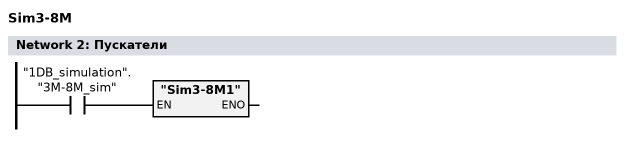
   RUNG wire#powerrail
      Contact( "1DB_simulation"."3M-8M_sim" )
      "Sim3-8M1"()
   END_RUNG
   // the same network as SCL:
   IF "1DB_simulation"."3M-8M_sim" THEN "Sim3-8M1"(); END_IF;
END_REGION
END_FUNCTION

FUNCTION "SimDym" : Void   // FC909, LAD
{ S7_Optimized_Access := 'TRUE' }
VERSION : 0.1
   VAR_TEMP
      trValue : Real;
      trValue_2 : Real;
      trValue_3 : Real;
   END_VAR
BEGIN

REGION Network 2: Скорость двигателя в %
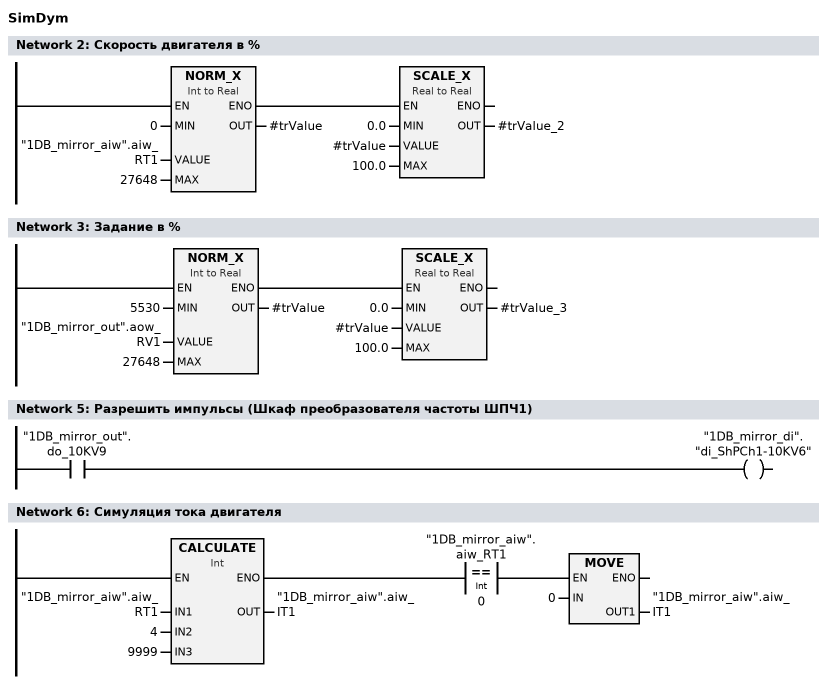
   RUNG wire#powerrail
      { S7_Templates := "[SrcType := Int, DestType := Real]" } Normalize(min := 0, value := "1DB_mirror_aiw".aiw_RT1, max := 27648, out => #trValue)
      { S7_Templates := "[SrcType := Real, DestType := Real]" } Scale(min := 0.0, value := #trValue, max := 100.0, out => #trValue_2)
   END_RUNG
   // the same network as SCL:
   #trValue := NORM_X(MIN := 0, VALUE := "1DB_mirror_aiw".aiw_RT1, MAX := 27648);
   #trValue_2 := SCALE_X(MIN := 0.0, VALUE := #trValue, MAX := 100.0);
END_REGION

REGION Network 3: Задание в %
   RUNG wire#powerrail
      { S7_Templates := "[SrcType := Int, DestType := Real]" } Normalize(min := 5530, value := "1DB_mirror_out".aow_RV1, max := 27648, out => #trValue)
      { S7_Templates := "[SrcType := Real, DestType := Real]" } Scale(min := 0.0, value := #trValue, max := 100.0, out => #trValue_3)
   END_RUNG
   // the same network as SCL:
   #trValue := NORM_X(MIN := 5530, VALUE := "1DB_mirror_out".aow_RV1, MAX := 27648);
   #trValue_3 := SCALE_X(MIN := 0.0, VALUE := #trValue, MAX := 100.0);
END_REGION

REGION Network 4 (SCL): Симуляция разгона и торможения
   //IF "1DB_mirror_out".do_1KV10 AND "1DB_mirror_out".do_1KV9
       //AND (NOT "HMI-Machinery".Dym.xSwitchAutoMode) THEN
   IF "1DB_mirror_out".aow_RV1 >0 THEN
       //IF #trValue_2 < "HMI-Machinery".Dym.rSpeedGoTo THEN
       IF #trValue_2 < #trValue_3 THEN
           "1DB_mirror_aiw".aiw_RT1 += 15;
       END_IF;
       IF #trValue_2 > #trValue_3 THEN
           "1DB_mirror_aiw".aiw_RT1 -= 19;
       END_IF;
   ELSE
       "1DB_mirror_aiw".aiw_RT1 := 0;
   END_IF;
END_REGION

REGION Network 5: Разрешить импульсы (Шкаф преобразователя частоты ШПЧ1)
   RUNG wire#powerrail
      Contact( "1DB_mirror_out".do_10KV9 )
      Coil( "1DB_mirror_di"."di_ShPCh1-10KV6" )
   END_RUNG
   // the same network as SCL:
   "1DB_mirror_di"."di_ShPCh1-10KV6" := "1DB_mirror_out".do_10KV9;
END_REGION

REGION Network 6: Симуляция тока двигателя
   RUNG wire#powerrail
      { S7_Templates := "SrcType := Int"; S7_Expression := "IN1/IN2 +IN3" } Calculate(in1 := "1DB_mirror_aiw".aiw_RT1, in2 := 4, in3 := 9999, out => "1DB_mirror_aiw".aiw_IT1)
      { S7_Templates := "SrcType := Int" } EQ_Contact(in1 := "1DB_mirror_aiw".aiw_RT1, in2 := 0)
      Move(in := 0, out1 => "1DB_mirror_aiw".aiw_IT1)
   END_RUNG
   // the same network as SCL:
   "1DB_mirror_aiw".aiw_IT1 := "1DB_mirror_aiw".aiw_RT1/4 +9999;
   IF "1DB_mirror_aiw".aiw_RT1 = 0 THEN "1DB_mirror_aiw".aiw_IT1 := 0; END_IF;
END_REGION
END_FUNCTION

FUNCTION "Sim2M1" : Void   // FC912, LAD
{ S7_Optimized_Access := 'TRUE' }
VERSION : 0.1
BEGIN

REGION Network 2: Пускатель КМ
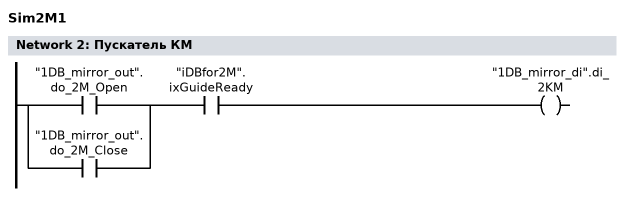
   RUNG wire#powerrail
      Contact( "1DB_mirror_out".do_2M_Open )
      wire#w1
      Contact( "iDBfor2M".ixGuideReady )
      Coil( "1DB_mirror_di".di_2KM )
   END_RUNG
   RUNG wire#powerrail
      Contact( "1DB_mirror_out".do_2M_Close )
   END_RUNG wire#w1
   // the same network as SCL:
   "1DB_mirror_di".di_2KM := ("1DB_mirror_out".do_2M_Open OR "1DB_mirror_out".do_2M_Close) AND "iDBfor2M".ixGuideReady;
END_REGION
END_FUNCTION

FUNCTION "Sim3-8M1" : Void   // FC913, LAD
{ S7_Optimized_Access := 'TRUE' }
VERSION : 0.1
BEGIN

REGION Network 2: Пускатель 3КМ1
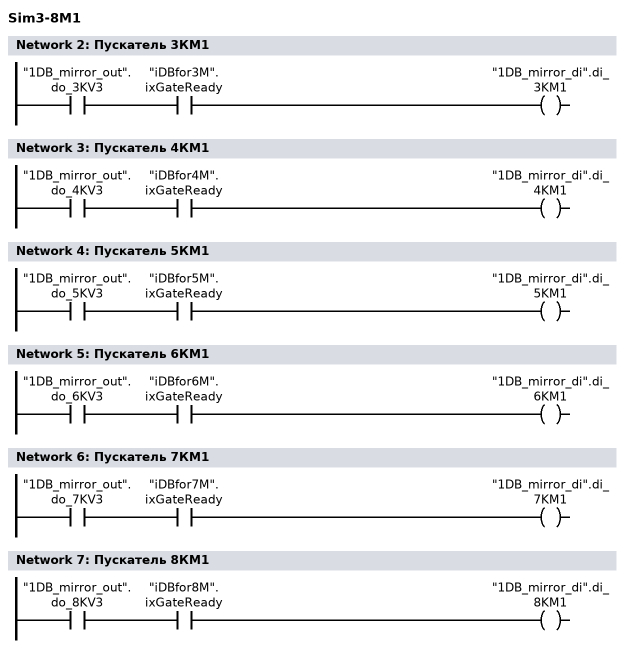
   RUNG wire#powerrail
      Contact( "1DB_mirror_out".do_3KV3 )
      Contact( "iDBfor3M".ixGateReady )
      Coil( "1DB_mirror_di".di_3KM1 )
   END_RUNG
   // the same network as SCL:
   "1DB_mirror_di".di_3KM1 := "1DB_mirror_out".do_3KV3 AND "iDBfor3M".ixGateReady;
END_REGION

REGION Network 3: Пускатель 4КМ1
   RUNG wire#powerrail
      Contact( "1DB_mirror_out".do_4KV3 )
      Contact( "iDBfor4M".ixGateReady )
      Coil( "1DB_mirror_di".di_4KM1 )
   END_RUNG
   // the same network as SCL:
   "1DB_mirror_di".di_4KM1 := "1DB_mirror_out".do_4KV3 AND "iDBfor4M".ixGateReady;
END_REGION

REGION Network 4: Пускатель 5КМ1
   RUNG wire#powerrail
      Contact( "1DB_mirror_out".do_5KV3 )
      Contact( "iDBfor5M".ixGateReady )
      Coil( "1DB_mirror_di".di_5KM1 )
   END_RUNG
   // the same network as SCL:
   "1DB_mirror_di".di_5KM1 := "1DB_mirror_out".do_5KV3 AND "iDBfor5M".ixGateReady;
END_REGION

REGION Network 5: Пускатель 6КМ1
   RUNG wire#powerrail
      Contact( "1DB_mirror_out".do_6KV3 )
      Contact( "iDBfor6M".ixGateReady )
      Coil( "1DB_mirror_di".di_6KM1 )
   END_RUNG
   // the same network as SCL:
   "1DB_mirror_di".di_6KM1 := "1DB_mirror_out".do_6KV3 AND "iDBfor6M".ixGateReady;
END_REGION

REGION Network 6: Пускатель 7КМ1
   RUNG wire#powerrail
      Contact( "1DB_mirror_out".do_7KV3 )
      Contact( "iDBfor7M".ixGateReady )
      Coil( "1DB_mirror_di".di_7KM1 )
   END_RUNG
   // the same network as SCL:
   "1DB_mirror_di".di_7KM1 := "1DB_mirror_out".do_7KV3 AND "iDBfor7M".ixGateReady;
END_REGION

REGION Network 7: Пускатель 8КМ1
   RUNG wire#powerrail
      Contact( "1DB_mirror_out".do_8KV3 )
      Contact( "iDBfor8M".ixGateReady )
      Coil( "1DB_mirror_di".di_8KM1 )
   END_RUNG
   // the same network as SCL:
   "1DB_mirror_di".di_8KM1 := "1DB_mirror_out".do_8KV3 AND "iDBfor8M".ixGateReady;
END_REGION
END_FUNCTION

FUNCTION "SimPower" : Void   // FC933, LAD
{ S7_Optimized_Access := 'TRUE' }
VERSION : 0.1
BEGIN

REGION Network 2: Симуляция сигналов электроснабжения DB112
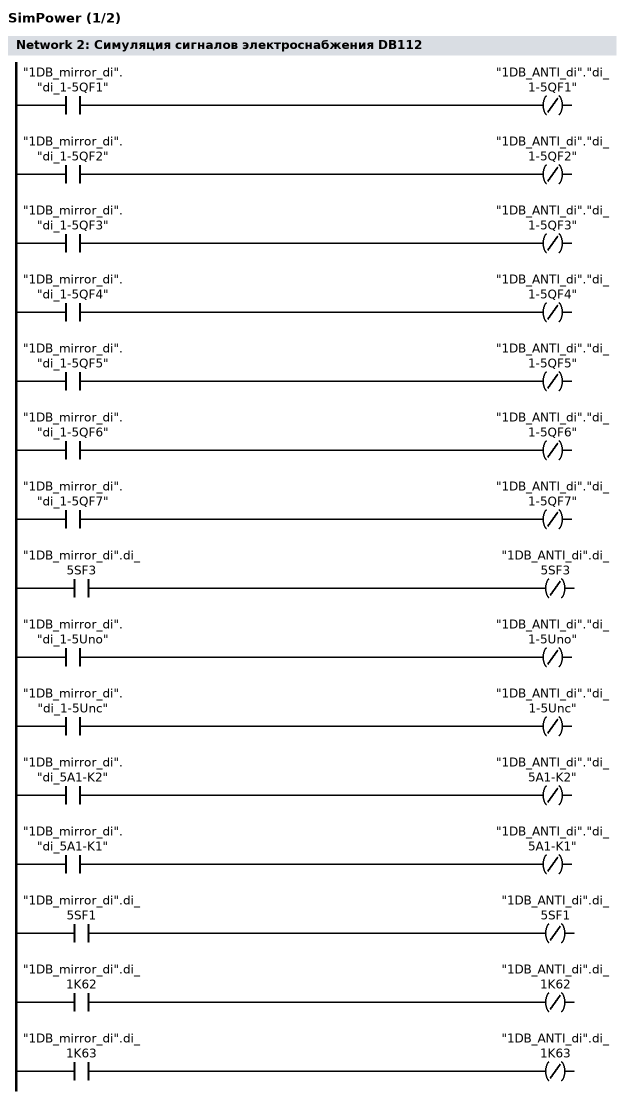
   RUNG wire#powerrail
      Contact( "1DB_mirror_di"."di_1-5QF1" )
      I_Coil( "1DB_ANTI_di"."di_1-5QF1" )
   END_RUNG
   RUNG wire#powerrail
      Contact( "1DB_mirror_di"."di_1-5QF2" )
      I_Coil( "1DB_ANTI_di"."di_1-5QF2" )
   END_RUNG
   RUNG wire#powerrail
      Contact( "1DB_mirror_di"."di_1-5QF3" )
      I_Coil( "1DB_ANTI_di"."di_1-5QF3" )
   END_RUNG
   RUNG wire#powerrail
      Contact( "1DB_mirror_di"."di_1-5QF4" )
      I_Coil( "1DB_ANTI_di"."di_1-5QF4" )
   END_RUNG
   RUNG wire#powerrail
      Contact( "1DB_mirror_di"."di_1-5QF5" )
      I_Coil( "1DB_ANTI_di"."di_1-5QF5" )
   END_RUNG
   RUNG wire#powerrail
      Contact( "1DB_mirror_di"."di_1-5QF6" )
      I_Coil( "1DB_ANTI_di"."di_1-5QF6" )
   END_RUNG
   RUNG wire#powerrail
      Contact( "1DB_mirror_di"."di_1-5QF7" )
      I_Coil( "1DB_ANTI_di"."di_1-5QF7" )
   END_RUNG
   RUNG wire#powerrail
      Contact( "1DB_mirror_di".di_5SF3 )
      I_Coil( "1DB_ANTI_di".di_5SF3 )
   END_RUNG
   RUNG wire#powerrail
      Contact( "1DB_mirror_di"."di_1-5Uno" )
      I_Coil( "1DB_ANTI_di"."di_1-5Uno" )
   END_RUNG
   RUNG wire#powerrail
      Contact( "1DB_mirror_di"."di_1-5Unc" )
      I_Coil( "1DB_ANTI_di"."di_1-5Unc" )
   END_RUNG
   RUNG wire#powerrail
      Contact( "1DB_mirror_di"."di_5A1-K2" )
      I_Coil( "1DB_ANTI_di"."di_5A1-K2" )
   END_RUNG
   RUNG wire#powerrail
      Contact( "1DB_mirror_di"."di_5A1-K1" )
      I_Coil( "1DB_ANTI_di"."di_5A1-K1" )
   END_RUNG
   RUNG wire#powerrail
      Contact( "1DB_mirror_di".di_5SF1 )
      I_Coil( "1DB_ANTI_di".di_5SF1 )
   END_RUNG
   RUNG wire#powerrail
      Contact( "1DB_mirror_di".di_1K62 )
      I_Coil( "1DB_ANTI_di".di_1K62 )
   END_RUNG
   RUNG wire#powerrail
      Contact( "1DB_mirror_di".di_1K63 )
      I_Coil( "1DB_ANTI_di".di_1K63 )
   END_RUNG
   // the same network as SCL:
   "1DB_ANTI_di"."di_1-5QF1" := NOT "1DB_mirror_di"."di_1-5QF1";
   "1DB_ANTI_di"."di_1-5QF2" := NOT "1DB_mirror_di"."di_1-5QF2";
   "1DB_ANTI_di"."di_1-5QF3" := NOT "1DB_mirror_di"."di_1-5QF3";
   "1DB_ANTI_di"."di_1-5QF4" := NOT "1DB_mirror_di"."di_1-5QF4";
   "1DB_ANTI_di"."di_1-5QF5" := NOT "1DB_mirror_di"."di_1-5QF5";
   "1DB_ANTI_di"."di_1-5QF6" := NOT "1DB_mirror_di"."di_1-5QF6";
   "1DB_ANTI_di"."di_1-5QF7" := NOT "1DB_mirror_di"."di_1-5QF7";
   "1DB_ANTI_di".di_5SF3 := NOT "1DB_mirror_di".di_5SF3;
   "1DB_ANTI_di"."di_1-5Uno" := NOT "1DB_mirror_di"."di_1-5Uno";
   "1DB_ANTI_di"."di_1-5Unc" := NOT "1DB_mirror_di"."di_1-5Unc";
   "1DB_ANTI_di"."di_5A1-K2" := NOT "1DB_mirror_di"."di_5A1-K2";
   "1DB_ANTI_di"."di_5A1-K1" := NOT "1DB_mirror_di"."di_5A1-K1";
   "1DB_ANTI_di".di_5SF1 := NOT "1DB_mirror_di".di_5SF1;
   "1DB_ANTI_di".di_1K62 := NOT "1DB_mirror_di".di_1K62;
   "1DB_ANTI_di".di_1K63 := NOT "1DB_mirror_di".di_1K63;
END_REGION

REGION Network 3: И далее
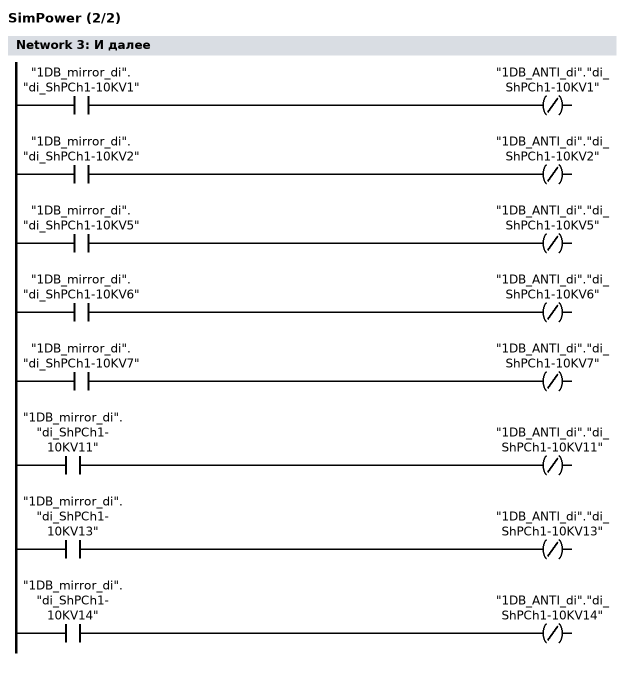
   RUNG wire#powerrail
      Contact( "1DB_mirror_di"."di_ShPCh1-10KV1" )
      I_Coil( "1DB_ANTI_di"."di_ShPCh1-10KV1" )
   END_RUNG
   RUNG wire#powerrail
      Contact( "1DB_mirror_di"."di_ShPCh1-10KV2" )
      I_Coil( "1DB_ANTI_di"."di_ShPCh1-10KV2" )
   END_RUNG
   RUNG wire#powerrail
      Contact( "1DB_mirror_di"."di_ShPCh1-10KV5" )
      I_Coil( "1DB_ANTI_di"."di_ShPCh1-10KV5" )
   END_RUNG
   RUNG wire#powerrail
      Contact( "1DB_mirror_di"."di_ShPCh1-10KV6" )
      I_Coil( "1DB_ANTI_di"."di_ShPCh1-10KV6" )
   END_RUNG
   RUNG wire#powerrail
      Contact( "1DB_mirror_di"."di_ShPCh1-10KV7" )
      I_Coil( "1DB_ANTI_di"."di_ShPCh1-10KV7" )
   END_RUNG
   RUNG wire#powerrail
      Contact( "1DB_mirror_di"."di_ShPCh1-10KV11" )
      I_Coil( "1DB_ANTI_di"."di_ShPCh1-10KV11" )
   END_RUNG
   RUNG wire#powerrail
      Contact( "1DB_mirror_di"."di_ShPCh1-10KV13" )
      I_Coil( "1DB_ANTI_di"."di_ShPCh1-10KV13" )
   END_RUNG
   RUNG wire#powerrail
      Contact( "1DB_mirror_di"."di_ShPCh1-10KV14" )
      I_Coil( "1DB_ANTI_di"."di_ShPCh1-10KV14" )
   END_RUNG
   // the same network as SCL:
   "1DB_ANTI_di"."di_ShPCh1-10KV1" := NOT "1DB_mirror_di"."di_ShPCh1-10KV1";
   "1DB_ANTI_di"."di_ShPCh1-10KV2" := NOT "1DB_mirror_di"."di_ShPCh1-10KV2";
   "1DB_ANTI_di"."di_ShPCh1-10KV5" := NOT "1DB_mirror_di"."di_ShPCh1-10KV5";
   "1DB_ANTI_di"."di_ShPCh1-10KV6" := NOT "1DB_mirror_di"."di_ShPCh1-10KV6";
   "1DB_ANTI_di"."di_ShPCh1-10KV7" := NOT "1DB_mirror_di"."di_ShPCh1-10KV7";
   "1DB_ANTI_di"."di_ShPCh1-10KV11" := NOT "1DB_mirror_di"."di_ShPCh1-10KV11";
   "1DB_ANTI_di"."di_ShPCh1-10KV13" := NOT "1DB_mirror_di"."di_ShPCh1-10KV13";
   "1DB_ANTI_di"."di_ShPCh1-10KV14" := NOT "1DB_mirror_di"."di_ShPCh1-10KV14";
END_REGION
END_FUNCTION

// folder: Simulation/SimGroup

FUNCTION "1FC_simAI" : Void   // FC990, SCL
{ S7_Optimized_Access := 'TRUE' }
VERSION : 0.1
   VAR_OUTPUT
      aiw : Int;
   END_VAR
   VAR_IN_OUT
      ioForSim : "uSim";
   END_VAR
   VAR_TEMP
      iTemp : Int;
      rTemp : Real;
   END_VAR
BEGIN

   //#rTemp := (315.0-197.0) * 223.0;
   //#iTemp := REAL_TO_INT(#rTemp);


   IF #ioForSim.config.up THEN
       IF #ioForSim.Value < 30000 THEN
           #ioForSim.Value += 237;
       END_IF;
   ELSE
       IF #ioForSim.config.down THEN
           IF #ioForSim.Value > -3000 THEN
               #ioForSim.Value -= 197;
           END_IF;
       ELSE
           #iTemp := "1DB_simTT".TForSim[#ioForSim.iCounter];
           #rTemp := INT_TO_REAL(#iTemp);
           #rTemp := #rTemp - #ioForSim.offset;
           #rTemp := #rTemp * #ioForSim.factor;
           #ioForSim.Value := REAL_TO_INT(#rTemp);
       END_IF;
   END_IF;
   #aiw := #ioForSim.Value;

   #ioForSim.iCounter += 1;
   IF #ioForSim.iCounter = 360 THEN
       #ioForSim.iCounter := 0;
   END_IF;
END_FUNCTION

FUNCTION "1FC_SimStartup" : Void   // FC991, LAD
{ S7_Optimized_Access := 'TRUE' }
VERSION : 0.1
BEGIN

REGION Network 2 (SCL): 1M
   //"1DB_mirror_di".di_1KV8 := TRUE;
   "1DB_mirror_di".di_1KM1_1KV8 := TRUE;
   "1DB_mirror_di".di_1KV6 := TRUE;

   //"1DB_mirror_aiw".aiw_TE102a := 2500;
END_REGION

REGION Network 3 (SCL): 2M
   "1DB_mirror_di".di_2KV1 := TRUE;
   "1DB_mirror_di".di_2KV4 := TRUE;
   "1DB_mirror_di".di_2KV3 := TRUE;
END_REGION

REGION Network 5 (SCL): 3M - 8M. Напряжение подано
   "1DB_mirror_di".di_3KV1 := TRUE;
   "1DB_mirror_di".di_4KV1 := TRUE;
   "1DB_mirror_di".di_5KV1 := TRUE;
   "1DB_mirror_di".di_6KV1 := TRUE;
   "1DB_mirror_di".di_7KV1 := TRUE;
   "1DB_mirror_di".di_8KV1 := TRUE;
END_REGION

REGION Network 6 (SCL): 3M - 8M. ДУ
   "1DB_mirror_di".di_3KV2 := TRUE;
   "1DB_mirror_di".di_4KV2 := TRUE;
   "1DB_mirror_di".di_5KV2 := TRUE;
   "1DB_mirror_di".di_6KV2 := TRUE;
   "1DB_mirror_di".di_7KV2 := TRUE;
   "1DB_mirror_di".di_8KV2 := TRUE;
END_REGION

REGION Network 7 (SCL): 3M - 8M. Автоматический режим
   "HMI-3M"."3M".xSwitchAutoMode := TRUE;
   "HMI-4M"."4M".xSwitchAutoMode := TRUE;
   "HMI-5M"."5M".xSwitchAutoMode := TRUE;
   "HMI-6M"."6M".xSwitchAutoMode := TRUE;
   "HMI-7M"."7M".xSwitchAutoMode := TRUE;
   "HMI-8M"."8M".xSwitchAutoMode := TRUE;
END_REGION

REGION Network 9 (SCL): Дымосос
   "1DB_mirror_di"."di_ShPCh1-10KV1" := TRUE;
   "1DB_mirror_di"."di_ShPCh1-10KV5" := TRUE;
   //"1DB_mirror_di"."di_ShPCh1-10KV6" := TRUE;    //Разрешить импульсы
   "1DB_mirror_di"."di_ShPCh1-10KV7" := TRUE;
   "1DB_mirror_di"."di_ShPCh1-10KV11" := TRUE;
   "1DB_mirror_di"."di_ShPCh1-10KV13" := TRUE;
   "HMI-Machinery".Dym.xReadyMaxStart := true;
END_REGION
END_FUNCTION

FUNCTION "1FC_simAI_RTD" : Void   // FC993, SCL
{ S7_Optimized_Access := 'TRUE' }
VERSION : 0.1
   VAR_OUTPUT
      aiw : Int;
   END_VAR
   VAR_IN_OUT
      ioForSim : "uSim";
   END_VAR
   VAR_TEMP
      iTemp : Int;
      rTemp : Real;
   END_VAR
BEGIN

   //#rTemp := (315.0-197.0) * 223.0;
   //#iTemp := REAL_TO_INT(#rTemp);


   IF #ioForSim.config.up THEN
       IF #ioForSim.Value < 30000 THEN
           #ioForSim.Value += 11;      //237;
       END_IF;
   ELSE
       IF #ioForSim.config.down THEN
           IF #ioForSim.Value > -3000 THEN
               #ioForSim.Value -= 9;   //197;
           END_IF;
       ELSE
           #iTemp := "1DB_simTT".TForSim[#ioForSim.iCounter];
           #rTemp := INT_TO_REAL(#iTemp);
           //#rTemp := #rTemp - #ioForSim.offset;
           //#rTemp := #rTemp * #ioForSim.factor;
           #ioForSim.Value := REAL_TO_INT(#rTemp);
       END_IF;
   END_IF;
   #aiw := #ioForSim.Value;

   #ioForSim.iCounter += 1;
   IF #ioForSim.iCounter = 360 THEN
       #ioForSim.iCounter := 0;
   END_IF;
END_FUNCTION

FUNCTION "1FC_simCummulative" : Void   // FC999, LAD
{ S7_Optimized_Access := 'TRUE' }
VERSION : 0.1
BEGIN

REGION Network 2: Симуляция для A1.02
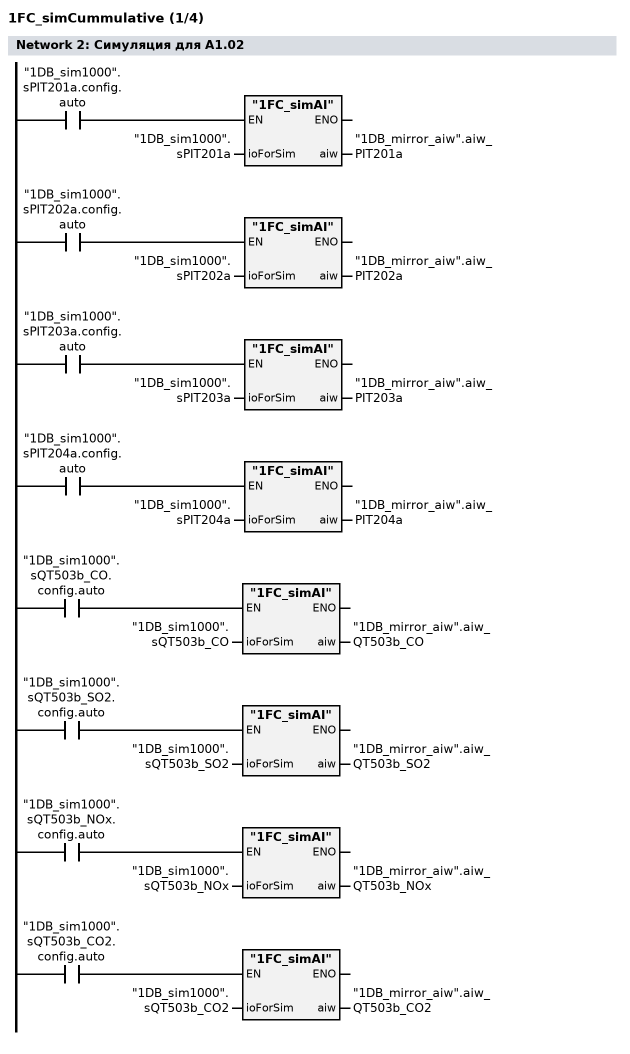
   RUNG wire#powerrail
      Contact( "1DB_sim1000".sPIT201a.config.auto )
      "1FC_simAI"(ioForSim := "1DB_sim1000".sPIT201a, aiw => "1DB_mirror_aiw".aiw_PIT201a)
   END_RUNG
   RUNG wire#powerrail
      Contact( "1DB_sim1000".sPIT202a.config.auto )
      "1FC_simAI"(ioForSim := "1DB_sim1000".sPIT202a, aiw => "1DB_mirror_aiw".aiw_PIT202a)
   END_RUNG
   RUNG wire#powerrail
      Contact( "1DB_sim1000".sPIT203a.config.auto )
      "1FC_simAI"(ioForSim := "1DB_sim1000".sPIT203a, aiw => "1DB_mirror_aiw".aiw_PIT203a)
   END_RUNG
   RUNG wire#powerrail
      Contact( "1DB_sim1000".sPIT204a.config.auto )
      "1FC_simAI"(ioForSim := "1DB_sim1000".sPIT204a, aiw => "1DB_mirror_aiw".aiw_PIT204a)
   END_RUNG
   RUNG wire#powerrail
      Contact( "1DB_sim1000".sQT503b_CO.config.auto )
      "1FC_simAI"(ioForSim := "1DB_sim1000".sQT503b_CO, aiw => "1DB_mirror_aiw".aiw_QT503b_CO)
   END_RUNG
   RUNG wire#powerrail
      Contact( "1DB_sim1000".sQT503b_SO2.config.auto )
      "1FC_simAI"(ioForSim := "1DB_sim1000".sQT503b_SO2, aiw => "1DB_mirror_aiw".aiw_QT503b_SO2)
   END_RUNG
   RUNG wire#powerrail
      Contact( "1DB_sim1000".sQT503b_NOx.config.auto )
      "1FC_simAI"(ioForSim := "1DB_sim1000".sQT503b_NOx, aiw => "1DB_mirror_aiw".aiw_QT503b_NOx)
   END_RUNG
   RUNG wire#powerrail
      Contact( "1DB_sim1000".sQT503b_CO2.config.auto )
      "1FC_simAI"(ioForSim := "1DB_sim1000".sQT503b_CO2, aiw => "1DB_mirror_aiw".aiw_QT503b_CO2)
   END_RUNG
   // the same network as SCL:
   IF "1DB_sim1000".sPIT201a.config.auto THEN
       "1FC_simAI"(ioForSim := "1DB_sim1000".sPIT201a, aiw => "1DB_mirror_aiw".aiw_PIT201a);
   END_IF;
   IF "1DB_sim1000".sPIT202a.config.auto THEN
       "1FC_simAI"(ioForSim := "1DB_sim1000".sPIT202a, aiw => "1DB_mirror_aiw".aiw_PIT202a);
   END_IF;
   IF "1DB_sim1000".sPIT203a.config.auto THEN
       "1FC_simAI"(ioForSim := "1DB_sim1000".sPIT203a, aiw => "1DB_mirror_aiw".aiw_PIT203a);
   END_IF;
   IF "1DB_sim1000".sPIT204a.config.auto THEN
       "1FC_simAI"(ioForSim := "1DB_sim1000".sPIT204a, aiw => "1DB_mirror_aiw".aiw_PIT204a);
   END_IF;
   IF "1DB_sim1000".sQT503b_CO.config.auto THEN
       "1FC_simAI"(ioForSim := "1DB_sim1000".sQT503b_CO, aiw => "1DB_mirror_aiw".aiw_QT503b_CO);
   END_IF;
   IF "1DB_sim1000".sQT503b_SO2.config.auto THEN
       "1FC_simAI"(ioForSim := "1DB_sim1000".sQT503b_SO2, aiw => "1DB_mirror_aiw".aiw_QT503b_SO2);
   END_IF;
   IF "1DB_sim1000".sQT503b_NOx.config.auto THEN
       "1FC_simAI"(ioForSim := "1DB_sim1000".sQT503b_NOx, aiw => "1DB_mirror_aiw".aiw_QT503b_NOx);
   END_IF;
   IF "1DB_sim1000".sQT503b_CO2.config.auto THEN
       "1FC_simAI"(ioForSim := "1DB_sim1000".sQT503b_CO2, aiw => "1DB_mirror_aiw".aiw_QT503b_CO2);
   END_IF;
END_REGION

REGION Network 3: Симуляция для A1.03
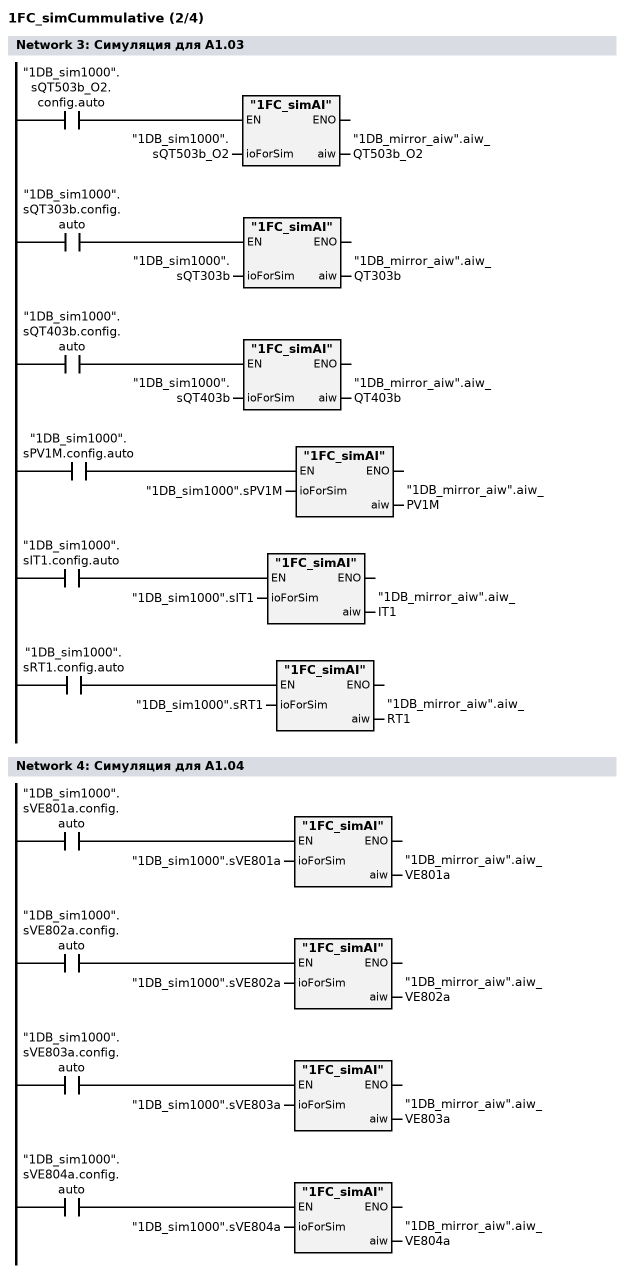
   RUNG wire#powerrail
      Contact( "1DB_sim1000".sQT503b_O2.config.auto )
      "1FC_simAI"(ioForSim := "1DB_sim1000".sQT503b_O2, aiw => "1DB_mirror_aiw".aiw_QT503b_O2)
   END_RUNG
   RUNG wire#powerrail
      Contact( "1DB_sim1000".sQT303b.config.auto )
      "1FC_simAI"(ioForSim := "1DB_sim1000".sQT303b, aiw => "1DB_mirror_aiw".aiw_QT303b)
   END_RUNG
   RUNG wire#powerrail
      Contact( "1DB_sim1000".sQT403b.config.auto )
      "1FC_simAI"(ioForSim := "1DB_sim1000".sQT403b, aiw => "1DB_mirror_aiw".aiw_QT403b)
   END_RUNG
   RUNG wire#powerrail
      Contact( "1DB_sim1000".sPV1M.config.auto )
      "1FC_simAI"(ioForSim := "1DB_sim1000".sPV1M, aiw => "1DB_mirror_aiw".aiw_PV1M)
   END_RUNG
   RUNG wire#powerrail
      Contact( "1DB_sim1000".sIT1.config.auto )
      "1FC_simAI"(ioForSim := "1DB_sim1000".sIT1, aiw => "1DB_mirror_aiw".aiw_IT1)
   END_RUNG
   RUNG wire#powerrail
      Contact( "1DB_sim1000".sRT1.config.auto )
      "1FC_simAI"(ioForSim := "1DB_sim1000".sRT1, aiw => "1DB_mirror_aiw".aiw_RT1)
   END_RUNG
   // the same network as SCL:
   IF "1DB_sim1000".sQT503b_O2.config.auto THEN
       "1FC_simAI"(ioForSim := "1DB_sim1000".sQT503b_O2, aiw => "1DB_mirror_aiw".aiw_QT503b_O2);
   END_IF;
   IF "1DB_sim1000".sQT303b.config.auto THEN
       "1FC_simAI"(ioForSim := "1DB_sim1000".sQT303b, aiw => "1DB_mirror_aiw".aiw_QT303b);
   END_IF;
   IF "1DB_sim1000".sQT403b.config.auto THEN
       "1FC_simAI"(ioForSim := "1DB_sim1000".sQT403b, aiw => "1DB_mirror_aiw".aiw_QT403b);
   END_IF;
   IF "1DB_sim1000".sPV1M.config.auto THEN
       "1FC_simAI"(ioForSim := "1DB_sim1000".sPV1M, aiw => "1DB_mirror_aiw".aiw_PV1M);
   END_IF;
   IF "1DB_sim1000".sIT1.config.auto THEN
       "1FC_simAI"(ioForSim := "1DB_sim1000".sIT1, aiw => "1DB_mirror_aiw".aiw_IT1);
   END_IF;
   IF "1DB_sim1000".sRT1.config.auto THEN
       "1FC_simAI"(ioForSim := "1DB_sim1000".sRT1, aiw => "1DB_mirror_aiw".aiw_RT1);
   END_IF;
END_REGION

REGION Network 4: Симуляция для A1.04
   RUNG wire#powerrail
      Contact( "1DB_sim1000".sVE801a.config.auto )
      "1FC_simAI"(ioForSim := "1DB_sim1000".sVE801a, aiw => "1DB_mirror_aiw".aiw_VE801a)
   END_RUNG
   RUNG wire#powerrail
      Contact( "1DB_sim1000".sVE802a.config.auto )
      "1FC_simAI"(ioForSim := "1DB_sim1000".sVE802a, aiw => "1DB_mirror_aiw".aiw_VE802a)
   END_RUNG
   RUNG wire#powerrail
      Contact( "1DB_sim1000".sVE803a.config.auto )
      "1FC_simAI"(ioForSim := "1DB_sim1000".sVE803a, aiw => "1DB_mirror_aiw".aiw_VE803a)
   END_RUNG
   RUNG wire#powerrail
      Contact( "1DB_sim1000".sVE804a.config.auto )
      "1FC_simAI"(ioForSim := "1DB_sim1000".sVE804a, aiw => "1DB_mirror_aiw".aiw_VE804a)
   END_RUNG
   // the same network as SCL:
   IF "1DB_sim1000".sVE801a.config.auto THEN
       "1FC_simAI"(ioForSim := "1DB_sim1000".sVE801a, aiw => "1DB_mirror_aiw".aiw_VE801a);
   END_IF;
   IF "1DB_sim1000".sVE802a.config.auto THEN
       "1FC_simAI"(ioForSim := "1DB_sim1000".sVE802a, aiw => "1DB_mirror_aiw".aiw_VE802a);
   END_IF;
   IF "1DB_sim1000".sVE803a.config.auto THEN
       "1FC_simAI"(ioForSim := "1DB_sim1000".sVE803a, aiw => "1DB_mirror_aiw".aiw_VE803a);
   END_IF;
   IF "1DB_sim1000".sVE804a.config.auto THEN
       "1FC_simAI"(ioForSim := "1DB_sim1000".sVE804a, aiw => "1DB_mirror_aiw".aiw_VE804a);
   END_IF;
END_REGION

REGION Network 5: Симуляция для A1.05
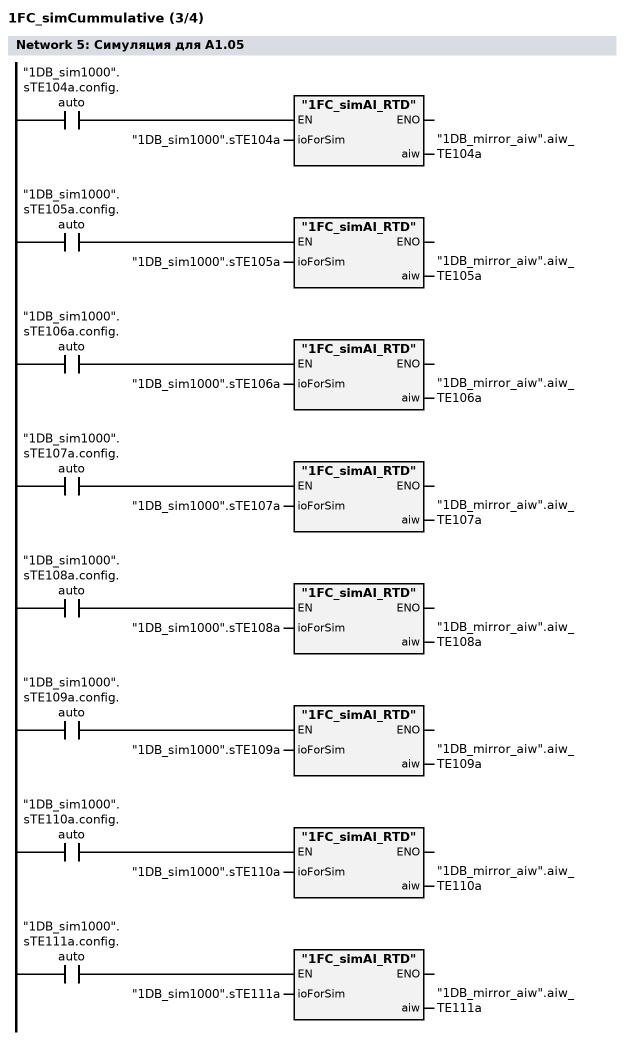
   RUNG wire#powerrail
      Contact( "1DB_sim1000".sTE104a.config.auto )
      "1FC_simAI_RTD"(ioForSim := "1DB_sim1000".sTE104a, aiw => "1DB_mirror_aiw".aiw_TE104a)
   END_RUNG
   RUNG wire#powerrail
      Contact( "1DB_sim1000".sTE105a.config.auto )
      "1FC_simAI_RTD"(ioForSim := "1DB_sim1000".sTE105a, aiw => "1DB_mirror_aiw".aiw_TE105a)
   END_RUNG
   RUNG wire#powerrail
      Contact( "1DB_sim1000".sTE106a.config.auto )
      "1FC_simAI_RTD"(ioForSim := "1DB_sim1000".sTE106a, aiw => "1DB_mirror_aiw".aiw_TE106a)
   END_RUNG
   RUNG wire#powerrail
      Contact( "1DB_sim1000".sTE107a.config.auto )
      "1FC_simAI_RTD"(ioForSim := "1DB_sim1000".sTE107a, aiw => "1DB_mirror_aiw".aiw_TE107a)
   END_RUNG
   RUNG wire#powerrail
      Contact( "1DB_sim1000".sTE108a.config.auto )
      "1FC_simAI_RTD"(ioForSim := "1DB_sim1000".sTE108a, aiw => "1DB_mirror_aiw".aiw_TE108a)
   END_RUNG
   RUNG wire#powerrail
      Contact( "1DB_sim1000".sTE109a.config.auto )
      "1FC_simAI_RTD"(ioForSim := "1DB_sim1000".sTE109a, aiw => "1DB_mirror_aiw".aiw_TE109a)
   END_RUNG
   RUNG wire#powerrail
      Contact( "1DB_sim1000".sTE110a.config.auto )
      "1FC_simAI_RTD"(ioForSim := "1DB_sim1000".sTE110a, aiw => "1DB_mirror_aiw".aiw_TE110a)
   END_RUNG
   RUNG wire#powerrail
      Contact( "1DB_sim1000".sTE111a.config.auto )
      "1FC_simAI_RTD"(ioForSim := "1DB_sim1000".sTE111a, aiw => "1DB_mirror_aiw".aiw_TE111a)
   END_RUNG
   // the same network as SCL:
   IF "1DB_sim1000".sTE104a.config.auto THEN
       "1FC_simAI_RTD"(ioForSim := "1DB_sim1000".sTE104a, aiw => "1DB_mirror_aiw".aiw_TE104a);
   END_IF;
   IF "1DB_sim1000".sTE105a.config.auto THEN
       "1FC_simAI_RTD"(ioForSim := "1DB_sim1000".sTE105a, aiw => "1DB_mirror_aiw".aiw_TE105a);
   END_IF;
   IF "1DB_sim1000".sTE106a.config.auto THEN
       "1FC_simAI_RTD"(ioForSim := "1DB_sim1000".sTE106a, aiw => "1DB_mirror_aiw".aiw_TE106a);
   END_IF;
   IF "1DB_sim1000".sTE107a.config.auto THEN
       "1FC_simAI_RTD"(ioForSim := "1DB_sim1000".sTE107a, aiw => "1DB_mirror_aiw".aiw_TE107a);
   END_IF;
   IF "1DB_sim1000".sTE108a.config.auto THEN
       "1FC_simAI_RTD"(ioForSim := "1DB_sim1000".sTE108a, aiw => "1DB_mirror_aiw".aiw_TE108a);
   END_IF;
   IF "1DB_sim1000".sTE109a.config.auto THEN
       "1FC_simAI_RTD"(ioForSim := "1DB_sim1000".sTE109a, aiw => "1DB_mirror_aiw".aiw_TE109a);
   END_IF;
   IF "1DB_sim1000".sTE110a.config.auto THEN
       "1FC_simAI_RTD"(ioForSim := "1DB_sim1000".sTE110a, aiw => "1DB_mirror_aiw".aiw_TE110a);
   END_IF;
   IF "1DB_sim1000".sTE111a.config.auto THEN
       "1FC_simAI_RTD"(ioForSim := "1DB_sim1000".sTE111a, aiw => "1DB_mirror_aiw".aiw_TE111a);
   END_IF;
END_REGION

REGION Network 6: Симуляция для A1.06
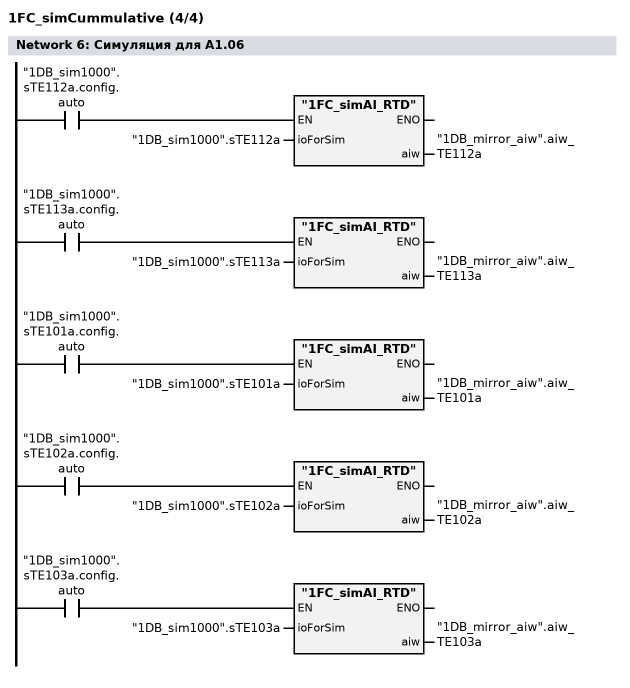
   RUNG wire#powerrail
      Contact( "1DB_sim1000".sTE112a.config.auto )
      "1FC_simAI_RTD"(ioForSim := "1DB_sim1000".sTE112a, aiw => "1DB_mirror_aiw".aiw_TE112a)
   END_RUNG
   RUNG wire#powerrail
      Contact( "1DB_sim1000".sTE113a.config.auto )
      "1FC_simAI_RTD"(ioForSim := "1DB_sim1000".sTE113a, aiw => "1DB_mirror_aiw".aiw_TE113a)
   END_RUNG
   RUNG wire#powerrail
      Contact( "1DB_sim1000".sTE101a.config.auto )
      "1FC_simAI_RTD"(ioForSim := "1DB_sim1000".sTE101a, aiw => "1DB_mirror_aiw".aiw_TE101a)
   END_RUNG
   RUNG wire#powerrail
      Contact( "1DB_sim1000".sTE102a.config.auto )
      "1FC_simAI_RTD"(ioForSim := "1DB_sim1000".sTE102a, aiw => "1DB_mirror_aiw".aiw_TE102a)
   END_RUNG
   RUNG wire#powerrail
      Contact( "1DB_sim1000".sTE103a.config.auto )
      "1FC_simAI_RTD"(ioForSim := "1DB_sim1000".sTE103a, aiw => "1DB_mirror_aiw".aiw_TE103a)
   END_RUNG
   // the same network as SCL:
   IF "1DB_sim1000".sTE112a.config.auto THEN
       "1FC_simAI_RTD"(ioForSim := "1DB_sim1000".sTE112a, aiw => "1DB_mirror_aiw".aiw_TE112a);
   END_IF;
   IF "1DB_sim1000".sTE113a.config.auto THEN
       "1FC_simAI_RTD"(ioForSim := "1DB_sim1000".sTE113a, aiw => "1DB_mirror_aiw".aiw_TE113a);
   END_IF;
   IF "1DB_sim1000".sTE101a.config.auto THEN
       "1FC_simAI_RTD"(ioForSim := "1DB_sim1000".sTE101a, aiw => "1DB_mirror_aiw".aiw_TE101a);
   END_IF;
   IF "1DB_sim1000".sTE102a.config.auto THEN
       "1FC_simAI_RTD"(ioForSim := "1DB_sim1000".sTE102a, aiw => "1DB_mirror_aiw".aiw_TE102a);
   END_IF;
   IF "1DB_sim1000".sTE103a.config.auto THEN
       "1FC_simAI_RTD"(ioForSim := "1DB_sim1000".sTE103a, aiw => "1DB_mirror_aiw".aiw_TE103a);
   END_IF;
END_REGION
END_FUNCTION